// TIA Portal V20 export
TYPE "typeScsMode"
// stored: Access Published, IsFailsafeCompliant true, Namespace Safety
   STRUCT
      Disabled : Bool;
      PendantReq : Bool;
      setup : Bool;
      auto : Bool;
      disable : Bool;
   END_STRUCT;
END_TYPE
